{attribute 'Tc2GvlVarNames'}
VAR_GLOBAL CONSTANT
	(*FiFo*)
	cMaxRowCMDFiFo			:INT := 50; (* Anzahl Maximal mögliche FiFo Zeilen *)
	cMaxScanIDs				:INT := 50;
END_VAR

(* stored: Version 1.1.0.1, ProductVersion 3.1.4024.15
   GVL GVL_HausBus_CONSTANT: Id {8ce5a7f4-2fc4-4c98-a646-25a6933cadc6} *)
